# EPICS substitutions: INSTRON/INSTRON-IOC-01App/Db/controls_channel.substitutions
file controls_channel.template {

pattern {PORT, P, CHAN, CHAN_UNITS, CHAN_NUM, CHAN_TOL, CHAN_EXP_TYPE }
{"\$(PORT)", "\$(P)", "POS", "mm", 1, 1, 0}
}
